Fanuc KAREL source: kx00022.KL

-- PROVISIONAL review KL for V770-1; original PC SHA256 e9be8c46184cc6595bec5edb240b00e75a144e8cd41bcd5425fe7869eef9e254
-- Incomplete behavior may be omitted. Consult companion uncertainty JSON. Do not deploy.
PROGRAM KX00022
%NOLOCKGROUP
VAR
  I : INTEGER
  J : INTEGER
  B : BOOLEAN
  F : FILE
  S : STRING[80]
-- UNRESOLVED_DECL P type=000102
-- UNRESOLVED_DECL BA type=002012
BEGIN
  -- UNRESOLVED_PC offsets 5-15; opcodes 9D,22,9D,33,35
  -- UNRESOLVED_PC offsets 20-35; opcodes 22,9D,33,34,23
  -- UNRESOLVED_PC offsets 40-44; opcodes 7F
END KX00022
